FUNCTION_BLOCK T_GripperMaintenanceMode EXTENDS T_NamedBase IMPLEMENTS I_PackMode
VAR
	_gripper : I_GripperModule;
END_VAR

METHOD Initialise
VAR_INPUT
	Gripper : I_GripperModule;
END_VAR
_gripper := Gripper;
END_METHOD

END_FUNCTION_BLOCK

(* stored: Version 1.1.0.1, ProductVersion 3.1.4024.12
   POU T_GripperMaintenanceMode: Id {c2fd17b7-5c19-4cd9-8362-9cd1c9e29854}, SpecialFunc None
   Method Initialise: Id {f69b160e-7628-4189-a9af-5b278fb8bfd4} *)
